(* CoDeSys 2.3 export: F_WRITE_LIFT_KEEL_CFG.EXP *)

(* POU FUN/PARAMETERS/F_WRITE_LIFT_KEEL_CFG, ST *)
FUNCTION F_WRITE_LIFT_KEEL_CFG : BOOL
VAR_INPUT
	sHead : STRING;
	wSize   :DWORD;
	pBuffer :POINTER TO BYTE;
END_VAR
VAR_IN_OUT
	wPos     : DWORD;
	stConfig : ST_LIFT_KEEL_CFG;
END_VAR
VAR
END_VAR
F_ADD_STRINGX3_TO_BUFFER( S1:= '$n#', S2:= sHead, S3:=' - Parameters:$n', wSize := wSize, pBuffer := pBuffer, wPos := wPos );

F_ADD_STRINGX4_TO_BUFFER( S1:= CONCAT(sHead, '_PMax_Up' ), S2:='$t', S3:= REAL_TO_STRING( stConfig.PMax_Up ), S4:='$n', wSize := wSize, pBuffer := pBuffer, wPos := wPos );
F_ADD_STRINGX4_TO_BUFFER( S1:= CONCAT(sHead, '_PMax_Dw' ), S2:='$t', S3:= REAL_TO_STRING( stConfig.PMax_Dw ), S4:='$n', wSize := wSize, pBuffer := pBuffer, wPos := wPos );
F_ADD_STRINGX4_TO_BUFFER( S1:= CONCAT(sHead, '_P500_Up' ), S2:='$t', S3:= REAL_TO_STRING( stConfig.P500_Up ), S4:='$n', wSize := wSize, pBuffer := pBuffer, wPos := wPos );
F_ADD_STRINGX4_TO_BUFFER( S1:= CONCAT(sHead, '_P500_Dw' ), S2:='$t', S3:= REAL_TO_STRING( stConfig.P500_Dw ), S4:='$n', wSize := wSize, pBuffer := pBuffer, wPos := wPos );
F_ADD_STRINGX4_TO_BUFFER( S1:= CONCAT(sHead, '_P144_F'  ), S2:='$t', S3:= REAL_TO_STRING( stConfig.P144_F  ), S4:='$n', wSize := wSize, pBuffer := pBuffer, wPos := wPos );
F_ADD_STRINGX4_TO_BUFFER( S1:= CONCAT(sHead, '_P144_S'  ), S2:='$t', S3:= REAL_TO_STRING( stConfig.P144_S  ), S4:='$n', wSize := wSize, pBuffer := pBuffer, wPos := wPos );

F_ADD_STRINGX4_TO_BUFFER( S1:= CONCAT(sHead, '_TgtP_Dw'  ), S2:='$t', S3:= REAL_TO_STRING( stConfig.TgtP_Dw  ), S4:='$n', wSize := wSize, pBuffer := pBuffer, wPos := wPos );
F_ADD_STRINGX4_TO_BUFFER( S1:= CONCAT(sHead, '_TgtLS_Up' ), S2:='$t', S3:= REAL_TO_STRING( stConfig.TgtLS_Up ), S4:='$n', wSize := wSize, pBuffer := pBuffer, wPos := wPos );
F_ADD_STRINGX4_TO_BUFFER( S1:= CONCAT(sHead, '_TgtLS_SUp' ), S2:='$t', S3:= REAL_TO_STRING( stConfig.TgtLS_SUp ), S4:='$n', wSize := wSize, pBuffer := pBuffer, wPos := wPos );
F_ADD_STRINGX4_TO_BUFFER( S1:= CONCAT(sHead, '_TgtLS_Dw' ), S2:='$t', S3:= REAL_TO_STRING( stConfig.TgtLS_Dw ), S4:='$n', wSize := wSize, pBuffer := pBuffer, wPos := wPos );

F_ADD_STRINGX4_TO_BUFFER( S1:= CONCAT(sHead, '_P_DB'     ), S2:='$t', S3:= REAL_TO_STRING( stConfig.P_DB     ), S4:='$n', wSize := wSize, pBuffer := pBuffer, wPos := wPos );
F_ADD_STRINGX4_TO_BUFFER( S1:= CONCAT(sHead, '_LS_DB'    ), S2:='$t', S3:= REAL_TO_STRING( stConfig.LS_DB    ), S4:='$n', wSize := wSize, pBuffer := pBuffer, wPos := wPos );
F_ADD_STRINGX4_TO_BUFFER( S1:= CONCAT(sHead, '_LS_Dist'  ), S2:='$t', S3:= REAL_TO_STRING( stConfig.LS_Dist  ), S4:='$n', wSize := wSize, pBuffer := pBuffer, wPos := wPos );

F_ADD_STRINGX4_TO_BUFFER( S1:= CONCAT(sHead, '_TimeMax'  ), S2:='$t', S3:= REAL_TO_STRING( stConfig.TimeMax  ), S4:='$n', wSize := wSize, pBuffer := pBuffer, wPos := wPos );
F_ADD_STRINGX4_TO_BUFFER( S1:= CONCAT(sHead, '_Delay_Dw' ), S2:='$t', S3:= REAL_TO_STRING( stConfig.Delay_Dw ), S4:='$n', wSize := wSize, pBuffer := pBuffer, wPos := wPos );

F_ADD_STRINGX4_TO_BUFFER( S1:= CONCAT(sHead, '_PP1'  ), S2:='$t', S3:= BOOL_TO_STRING( stConfig.PP1 ), S4:='$n', wSize := wSize, pBuffer := pBuffer, wPos := wPos );
F_ADD_STRINGX4_TO_BUFFER( S1:= CONCAT(sHead, '_PP2'  ), S2:='$t', S3:= BOOL_TO_STRING( stConfig.PP2 ), S4:='$n', wSize := wSize, pBuffer := pBuffer, wPos := wPos );
F_ADD_STRINGX4_TO_BUFFER( S1:= CONCAT(sHead, '_HP1'  ), S2:='$t', S3:= BOOL_TO_STRING( stConfig.HP1 ), S4:='$n', wSize := wSize, pBuffer := pBuffer, wPos := wPos );
F_ADD_STRINGX4_TO_BUFFER( S1:= CONCAT(sHead, '_HP2'  ), S2:='$t', S3:= BOOL_TO_STRING( stConfig.HP2 ), S4:='$n', wSize := wSize, pBuffer := pBuffer, wPos := wPos );
F_ADD_STRINGX4_TO_BUFFER( S1:= CONCAT(sHead, '_HP3'  ), S2:='$t', S3:= BOOL_TO_STRING( stConfig.HP3 ), S4:='$n', wSize := wSize, pBuffer := pBuffer, wPos := wPos );
END_FUNCTION
